FUNCTION_BLOCK PUBLIC FB_FactoryIO_ModbusTCP_Read
VAR_INPUT
	// **** Configuration en fonction de la configuration FactoryIO
	sIPAddr : STRING[15]:='127.0.0.1'; // '127.0.0.1'
	nTCPPort : UINT:=505; // 505
	nUnitID : BYTE:=255; // 255	
END_VAR

VAR_OUTPUT
	bBusy: BOOL;
	bError: BOOL;
	// *** Configuration des array en fonction de la configuration FactoryIO
	InputReg : ARRAY [0..7] OF INT; // ex. input register 8 [0..7] pour les mesures analogiques
	// Inputs traités
	bInput1 : ARRAY [0..15] OF BOOL;
	bInput2 : ARRAY [0..15] OF BOOL;
	
END_VAR
	
VAR
	// Instances
	fb_MBReadInputs : FB_MBReadInputs; // Instance de la fonction FB_MBReadInputs de la lib Tc2_ModbusSrv
	fb_MBReadInputRegs : FB_MBReadInputRegs;
	
	fb_Word_To_Bool : FB_Word_To_Bool; // Instance commune
	fb_Bool_To_Word: FB_Bool_To_Word ; // Instance commune
	
	// *** Configuration des array en fonction de la configuration FactoryIO
	Input : ARRAY [0..1] OF WORD; // ex. input digital 16 [0..0] /  input digital 32 [0..1]
	
	// Busy Error interne à la fonciton
	bBusyInput: ARRAY [1..2] OF BOOL;
	bErrorInput: ARRAY [1..2] OF BOOL;

END_VAR

// Traitement des bool représentant les inputs
fb_Word_To_Bool(inWord := Input[0],
				outArrayOfBool => bInput1);
fb_Word_To_Bool(inWord := Input[1],
				outArrayOfBool => bInput2);
				
			

// Busy si au moins 1 busy
IF bBusyInput[1] OR bBusyInput[2] THEN
	bBusy := 1;
ELSE
	bBusy := 0;
END_IF

// Error si au moins 1 busy
IF bErrorInput[1] OR bErrorInput[2] THEN
	bError := 1;
ELSE
	bError := 0;
END_IF

METHOD MappingInput
VAR_INPUT
END_VAR
// Exercice 1
E_BoutonMarche := FIO_Input1[0];
E_Capteur := FIO_Input1[1];
E_BoutonAvancer := FIO_Input1[2];
END_METHOD

METHOD PUBLIC ReadInput
fb_MBReadInputs(
	sIPAddr := sIPAddr,
	nTCPPort := nTCPPort,
	nUnitID := nUnitID,
	nQuantity := SIZEOF(Input)*8, // Nombre de bits à lire SIZEOF(nb byte * bits dans 1 byte)
	nMBAddr := 0,
	cbLength := SIZEOF(Input),
	pDestAddr := ADR(Input),
	bExecute := TRUE,
	tTimeout := T#1S,
	bBusy => bBusyInput[1],
	bError => bErrorInput[1],
	nErrId => ,
	cbRead => ,
 );
fb_MBReadInputs(bExecute := FALSE);
END_METHOD

METHOD PUBLIC ReadInputRegister
fb_MBReadInputRegs(
	sIPAddr := sIPAddr,
	nTCPPort := nTCPPort,
	nUnitID := nUnitID,
	nQuantity := SIZEOF(InputReg)/2,
	nMBAddr := 0,
	cbLength := SIZEOF(InputReg),
	pDestAddr := ADR(InputReg),
	bExecute := TRUE,
	tTimeout := T#1S,
	bBusy => bBusyInput[2],
	bError => bErrorInput[2],
	nErrId => ,
	cbRead => ,
 );
fb_MBReadInputRegs(bExecute := FALSE);
END_METHOD

END_FUNCTION_BLOCK

(* stored: Version 1.1.0.1, ProductVersion 3.1.4024.11
   POU FB_FactoryIO_ModbusTCP_Read: Id {ef99659b-bb0e-494d-8cf7-6072e7c46a5c}, SpecialFunc None
   Method MappingInput: Id {cdba02c1-7fcc-49d0-8394-7d19715afbb4}
   Method ReadInput: Id {114b7d6d-1641-41a1-9a37-c80540c5b291}
   Method ReadInputRegister: Id {49627f2a-4539-4976-b388-686bcf311a5b} *)
